// TIA Portal V17 export
// export: Created 2023-05-07T12:12:22.0811285Z, ExportSetting WithDefaults, DisplayName Totally Integrated Automation Portal, DisplayVersion V17, DisplayName TIA Portal Openness, DisplayVersion V17, DisplayName TIA Portal Version Control Interface, DisplayVersion V17, DisplayName TIA Portal Test Suite Advanced, DisplayVersion V17, DisplayName STEP 7 Professional, DisplayVersion V17, DisplayName SIMATIC Energy Suite, DisplayVersion V17, DisplayName STEP 7 Safety, DisplayVersion V17, DisplayName WinCC Professional, DisplayVersion V17
DATA_BLOCK "PID_DB"   // DB2
VERSION : 0.1
// stored: AutoNumber true, InstanceOfName PID, InstanceOfType FB
"PID"
   // VAR_INPUT
   //    SP : Real;
   //    PV : Real;
   //    MV : Real;
   //    kp : Real;
   //    ki : Real;
   //    kd : Real;
   // END_VAR
   // VAR_OUTPUT
   //    MV_PID : Real;
   // END_VAR
   // VAR
   //    ep : Array[0..1] of Real;
   //    de : Real;
   //    suma_ep : Real;
   // END_VAR
BEGIN
END_DATA_BLOCK
